// TIA Portal project "2M4" (V16)

(* hardware
DEVICE "S7-1200 station_1"  S7-1200 Station
   slot 0: "Rack_0"  S7-1200 Rack  Rack  V1.0
   slot 1: "PLC_1"  CPU 1212C AC/DC/Rly  6ES7 212-1BE40-0XB0  V4.4
*)

// ===== PLC "PLC_1"  CPU 1212C AC/DC/Rly =====

VAR_GLOBAL   // PLC tag table "Default tag table"
   "START" AT %I0.1 : Bool;
   "STOP" AT %I0.2 : Bool;
   "MOTOR1" AT %Q0.0 : Bool;
   "MOTOR2" AT %Q0.1 : Bool;
   "CM" AT %M0.0 : Bool;
   "TM1" AT %M0.1 : Bool;
   "TM2" AT %M0.2 : Bool;
   "T1ON" AT %M0.3 : Bool;
   "T2ON" AT %M0.4 : Bool;
   "Tag_1" AT %M0.7 : Bool;
   "Tag_2" AT %M0.5 : Bool;
   "Tag_3" AT %M0.6 : Bool;
   "Tag_4" AT %M1.2 : Bool;
   "Tag_5" AT %M1.7 : Bool;
   "Tag_6" AT %M1.5 : Bool;
END_VAR

// folder: System blocks/Program resources

DATA_BLOCK "COUNTER"   // DB1
{ S7_Optimized_Access := 'TRUE' }
AUTHOR : Simatic
FAMILY : IEC
NAME : CNTR
VERSION : 1.0
// stored: InstanceOfName IEC_COUNTER
"IEC_COUNTER"
BEGIN
END_DATA_BLOCK

DATA_BLOCK "TIMER1"   // DB2
{ S7_Optimized_Access := 'TRUE' }
AUTHOR : Simatic
FAMILY : IEC
NAME : IEC_TMR
VERSION : 1.0
// stored: InstanceOfName IEC_TIMER
"IEC_TIMER"
BEGIN
END_DATA_BLOCK

DATA_BLOCK "TIMER2"   // DB3
{ S7_Optimized_Access := 'TRUE' }
AUTHOR : Simatic
FAMILY : IEC
NAME : IEC_TMR
VERSION : 1.0
// stored: InstanceOfName IEC_TIMER
"IEC_TIMER"
BEGIN
END_DATA_BLOCK

// folder: (top level)

ORGANIZATION_BLOCK "Main"   // OB1, LAD, ProgramCycle
TITLE = "Main Program Sweep (Cycle)"
{ S7_Optimized_Access := 'TRUE' }
VERSION : 0.1
   VAR_INPUT
      Initial_Call : Bool;   // Initial call of this OB
      Remanence : Bool;   // =True, if remanent data are available
   END_VAR
   VAR_TEMP   // added for the SCL form of the ladder/FBD networks
      _w1 : Bool;
   END_VAR
BEGIN

REGION Network 1
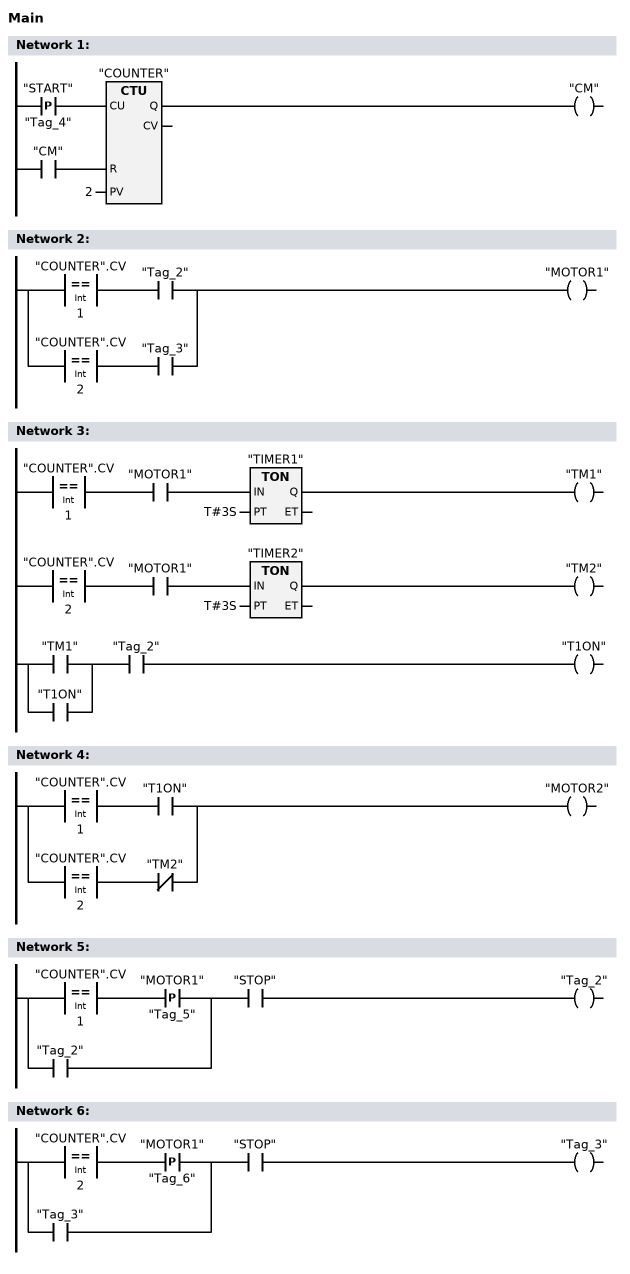
   #_w1 := "START" AND NOT "Tag_4";   // rising edge of "START"
   "Tag_4" := "START";
   "COUNTER".CTU(CU := #_w1, R := "CM", PV := 2);
   "CM" := "COUNTER".Q;
END_REGION

REGION Network 2
   RUNG wire#powerrail
      { S7_Templates := "SrcType := Int" } EQ_Contact(in1 := "COUNTER".CV, in2 := 1)
      Contact( "Tag_2" )
      wire#w1
      Coil( "MOTOR1" )
   END_RUNG
   RUNG wire#powerrail
      { S7_Templates := "SrcType := Int" } EQ_Contact(in1 := "COUNTER".CV, in2 := 2)
      Contact( "Tag_3" )
   END_RUNG wire#w1
   // the same network as SCL:
   "MOTOR1" := (("COUNTER".CV = 1) AND "Tag_2") OR (("COUNTER".CV = 2) AND "Tag_3");
END_REGION

REGION Network 3
   "TIMER1".TON(IN := ("COUNTER".CV = 1) AND "MOTOR1", PT := T#3S);
   "TM1" := "TIMER1".Q;
   "TIMER2".TON(IN := ("COUNTER".CV = 2) AND "MOTOR1", PT := T#3S);
   "TM2" := "TIMER2".Q;
   "T1ON" := ("TM1" OR "T1ON") AND "Tag_2";
END_REGION

REGION Network 4
   RUNG wire#powerrail
      { S7_Templates := "SrcType := Int" } EQ_Contact(in1 := "COUNTER".CV, in2 := 1)
      Contact( "T1ON" )
      wire#w1
      Coil( "MOTOR2" )
   END_RUNG
   RUNG wire#powerrail
      { S7_Templates := "SrcType := Int" } EQ_Contact(in1 := "COUNTER".CV, in2 := 2)
      I_Contact( "TM2" )
   END_RUNG wire#w1
   // the same network as SCL:
   "MOTOR2" := (("COUNTER".CV = 1) AND "T1ON") OR (("COUNTER".CV = 2) AND NOT "TM2");
END_REGION

REGION Network 5
   RUNG wire#powerrail
      { S7_Templates := "SrcType := Int" } EQ_Contact(in1 := "COUNTER".CV, in2 := 1)
      P_Contact(operand := "MOTOR1", bit := "Tag_5")
      wire#w1
      Contact( "STOP" )
      Coil( "Tag_2" )
   END_RUNG
   RUNG wire#powerrail
      Contact( "Tag_2" )
   END_RUNG wire#w1
   // the same network as SCL:
   #_w1 := ("COUNTER".CV = 1) AND "MOTOR1" AND NOT "Tag_5";   // rising edge of "MOTOR1"
   "Tag_5" := "MOTOR1";
   "Tag_2" := (#_w1 OR "Tag_2") AND "STOP";
END_REGION

REGION Network 6
   RUNG wire#powerrail
      { S7_Templates := "SrcType := Int" } EQ_Contact(in1 := "COUNTER".CV, in2 := 2)
      P_Contact(operand := "MOTOR1", bit := "Tag_6")
      wire#w1
      Contact( "STOP" )
      Coil( "Tag_3" )
   END_RUNG
   RUNG wire#powerrail
      Contact( "Tag_3" )
   END_RUNG wire#w1
   // the same network as SCL:
   #_w1 := ("COUNTER".CV = 2) AND "MOTOR1" AND NOT "Tag_6";   // rising edge of "MOTOR1"
   "Tag_6" := "MOTOR1";
   "Tag_3" := (#_w1 OR "Tag_3") AND "STOP";
END_REGION
END_ORGANIZATION_BLOCK